{attribute 'GeneratedUsingTerminal: EL4012-0000-0018'}
{attribute addProperty BoxType "EL4012-0000-0018"}
{attribute addProperty Id "EtcSlaveTerminalBaseAO_Output_Channel_1AT %Q*AO_Output_Channel_BA7EBB7C2AO_Output_Channel_2AT %Q*AO_Output_Channel_BA7EBB7C2WcStateAT %I*WcState_0B2B16F91InfoDataAT %I*InfoData_32EB74EA10"}
{attribute addProperty CRC "910503028"}
{attribute addProperty Size "15"}
TYPE EL4012_36452C74 EXTENDS EtcSlaveTerminalBase :
STRUCT
	{attribute addProperty Name "AO_Output_Channel_1"}
	AO_Output_Channel_1 : AO_Output_Channel_BA7EBB7C;
	{attribute addProperty Name "AO_Output_Channel_2"}
	AO_Output_Channel_2 : AO_Output_Channel_BA7EBB7C;
	{attribute addProperty Name "WcState"}
	WcState : WcState_0B2B16F9;
	{attribute addProperty Name "InfoData"}
	InfoData : InfoData_32EB74EA;
END_STRUCT
END_TYPE

(* stored: Version 1.2.0.0, ProductVersion 3.1.4024.9
   DUT EL4012_36452C74: Id {a87df7f1-0fbf-48be-814e-54326bcdaf89} *)
